Universal Robots PolyScope program: huy.urp

Program huy (installation=default directory=/ursim/programs createdIn=5.25.1 lastSavedIn=5.25.1 robotSerialNumber=20195399999)
Calibrated DH parameters: a=[0, -0.24355, -0.2132, 0, 0, 0]; d=[0.15185, 0, 0, 0.13105, 0.08535, 0.0921]; alpha=[1.570796, 0, 0, 1.570796, -1.570796, 0]; deltaTheta=[0, 0, 0, 0, 0, 0]
InitVariablesNode
Robot Program (runOnlyOnce=false)
  URCap External Control (External Control, FZI Research Center for Information Technology)
